SUBAPPLICATION Uebung_224b (* Standard IEC 61131-3 FB_CTUD_ULINT (Vor-/Rückwärtszähler, ULINT) mit Terminal-Ausgabe (PHYS_LREAL) *)
  (* Standard: 61131-3; Description: Copyright (c) 2026 Meisterschulen am Ostbahnhof This program and the accompanying materials are made available under the terms of the Eclipse Public License 2.0 which is available at https://www.eclipse.org/legal/epl-2.0/ SPDX-License-Identifier: EPL-2.0 *)
  (* Version 1.1, 2026-04-21, Franz Höpfinger, Meisterschulen am Ostbahnhof, Added terminal output for counter value (PHYS_LREAL + Converter) *)
  (* Version 1.0, 2026-04-20, Franz Höpfinger, Meisterschulen am Ostbahnhof, initial API and implementation (IEC 61131-3 version) *)
  PACKAGE Uebungen;
  IMPORT Uebungen::const::UT::DefaultPool_Numeric::OutputNumber_N3_N;
  IMPORT logiBUS::io::DI::logiBUS_DI::Input_I1;
  IMPORT logiBUS::io::DI::logiBUS_DI::Input_I2;
  IMPORT logiBUS::io::DI::logiBUS_DI::Input_I3;
  IMPORT logiBUS::io::DI::logiBUS_DI::Input_I4;
  IMPORT logiBUS::io::DQ::logiBUS_DO::Output_Q1;
  IMPORT logiBUS::io::DQ::logiBUS_DO::Output_Q2;
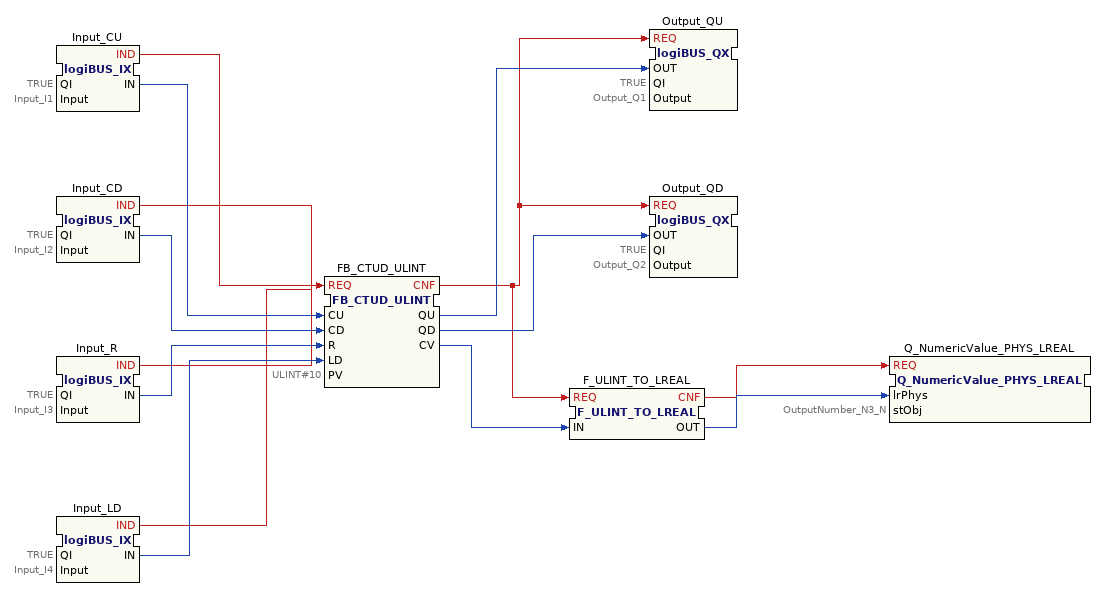
  (* hier gegebenenfalls (einen oder zwei) E_D_FF einbauen, damit die Events reduziert werden. *)
  FBS
    FB_CTUD_ULINT : iec61131::counters::FB_CTUD_ULINT(PV := ULINT#10);
    Input_CU : logiBUS::io::DI::logiBUS_IX(QI := TRUE, Input := Input_I1);
    Input_CD : logiBUS::io::DI::logiBUS_IX(QI := TRUE, Input := Input_I2);
    Input_R : logiBUS::io::DI::logiBUS_IX(QI := TRUE, Input := Input_I3);
    Input_LD : logiBUS::io::DI::logiBUS_IX(QI := TRUE, Input := Input_I4);
    Output_QU : logiBUS::io::DQ::logiBUS_QX(QI := TRUE, Output := Output_Q1);
    Output_QD : logiBUS::io::DQ::logiBUS_QX(QI := TRUE, Output := Output_Q2);
    F_ULINT_TO_LREAL : iec61131::conversion::F_ULINT_TO_LREAL;
    Q_NumericValue_PHYS_LREAL : isobus::UT::Q::Q_NumericValue_PHYS_LREAL(stObj := OutputNumber_N3_N);
  END_FBS
  EVENT_CONNECTIONS
    Input_CU.IND TO FB_CTUD_ULINT.REQ;
    Input_CD.IND TO FB_CTUD_ULINT.REQ;
    Input_R.IND TO FB_CTUD_ULINT.REQ;
    Input_LD.IND TO FB_CTUD_ULINT.REQ;
    FB_CTUD_ULINT.CNF TO Output_QU.REQ;
    FB_CTUD_ULINT.CNF TO Output_QD.REQ;
    FB_CTUD_ULINT.CNF TO F_ULINT_TO_LREAL.REQ;
    F_ULINT_TO_LREAL.CNF TO Q_NumericValue_PHYS_LREAL.REQ;
  END_CONNECTIONS
  DATA_CONNECTIONS
    Input_CU.IN TO FB_CTUD_ULINT.CU;
    Input_CD.IN TO FB_CTUD_ULINT.CD;
    Input_R.IN TO FB_CTUD_ULINT.R;
    Input_LD.IN TO FB_CTUD_ULINT.LD;
    FB_CTUD_ULINT.QU TO Output_QU.OUT;
    FB_CTUD_ULINT.QD TO Output_QD.OUT;
    FB_CTUD_ULINT.CV TO F_ULINT_TO_LREAL.IN;
    F_ULINT_TO_LREAL.OUT TO Q_NumericValue_PHYS_LREAL.lrPhys;
  END_CONNECTIONS
END_SUBAPPLICATION
